FUNCTION_BLOCK FB_DiscreteValve EXTENDS FB_Actor2Point
VAR_INPUT
END_VAR
VAR_OUTPUT
END_VAR
VAR
	//default parameters
	localDefaultParameters : ST_DiscreteValveDefaultParameters;	

	//I/O Links
	bSetStatusOn_OUT 	AT %Q* : BOOL := FALSE;
	bStatusOn_IN		AT %I* : BOOL := FALSE; //True if valve is (actual) open
END_VAR

SelectControlMode();

METHOD SetState_BI_BO : BOOL
VAR_INPUT
END_VAR
VAR
END_VAR
//control state
IF localDefaultParameters.bFeedbackSignal = TRUE THEN //Use feedback signal if possible
	controlState.bStatusOn := bStatusOn_IN;
	bStatusOn := bStatusOn_IN;
END_IF;

//output
bSetStatusOn_OUT := bSetStatusOn;
END_METHOD

PROPERTY ST_DefaultParameters : REFERENCE TO ST_DiscreteValveDefaultParameters
SET
localDefaultParameters := ST_DefaultParameters;
END_SET
END_PROPERTY

END_FUNCTION_BLOCK

(* stored: Version 1.1.0.1, ProductVersion 3.1.4024.9
   POU FB_DiscreteValve: Id {7c2d056e-b7a5-47e0-8780-c9ad927c4f52}, SpecialFunc None
   Method SetState_BI_BO: Id {0e571675-b07a-4d0e-a5bb-9e330e7c5235}
   Property ST_DefaultParameters: Id {8d33a13c-5650-4ddc-aac7-e5707e8c1b8d}
   Set Set: Id {33d3ed96-b96e-4f0c-89d2-38cef331df44} *)
